// TwinCAT 3 PLC project Tc_SystemCx
// Title: Tc_SystemCx
// Company: NewEngineer
// Author: https://github.com/phucpha
// ProjectVersion: 0.0.0.1
// Description: This library expand of Tc2_systemCx
// ProgramVersion: 3.1.4024.0
// libraries:
//   Tc2_SystemCX, * (Beckhoff Automation GmbH)
//   Tc2_Utilities, * (Beckhoff Automation GmbH)
//   Tc3_Module, * (Beckhoff Automation GmbH)
// project tree:
//   / PlcTask.TcTTO
//   POUs/Cx70xx/ FB_Cx7_Read_EEPROM_CFIRM_KEY.TcPOU
//   Version/ Global_Version.TcGVL
// real-time tasks:
//   TASK PlcTask: cycle T#10ms, priority 20, ADS port 350

CONFIGURATION Tc_SystemCx
    RESOURCE PLC ON TwinCAT3
        TASK PlcTask(INTERVAL := T#10ms, PRIORITY := 20);
    END_RESOURCE
END_CONFIGURATION

// ---- Version/Global_Version.TcGVL
{attribute 'TcGenerated'}
{attribute 'no-analysis'}
{attribute 'linkalways'}
// This function has been automatically generated from the project information.
VAR_GLOBAL CONSTANT
	{attribute 'const_non_replaced'}
	stLibVersion_Tc_SystemCx : ST_LibVersion := (iMajor := 0, iMinor := 0, iBuild := 0, iRevision := 1, nFlags := 0, sVersion := '0.0.0.1');
END_VAR

// ---- POUs/Cx70xx/FB_Cx7_Read_EEPROM_CFIRM_KEY.TcPOU
{attribute 'hide_all_locals'}
FUNCTION_BLOCK FB_Cx7_Read_EEPROM_CFIRM_KEY
VAR_INPUT
	psKey: POINTER TO STRING(31);
END_VAR

VAR
	arrEEPRomRead : ARRAY [0..nSizeOfHASH_SHA512-1] OF BYTE;
	arrbHashGen : ARRAY [0..nSizeOfHASH_SHA512-1] OF BYTE;// Shouldn't edit it
// EEPROM
	bBusy            : BOOL;         // FB is working
    bEEpromError     : BOOL;         // FB has an Error
    nErrorID         : UDINT;        (* Error Code
    If nErrorID=DEVICE_INVALIDACCESS the EEPROM write cycles reached max. value. 
    If nErrorID=DEVICE_INVALIDPARM the given pointer parameter is invalid/null. 
    If nErrorID=DEVICE_INVALIDSIZE the given buffer size is too small or too big.
    If nErrorID=DEVICE_SRVNOTSUPP probably the image version need to be updated to support this feature. *)
    nDataSizeEEPROM  : UINT;         // current size of (read) EEPROM data in bytes (max.120 Bytes)
    nWritesCycles    : UINT;         // already performed EEPROM write cycles (maximum possible = 200)
	eRead 			 : UINT;
	fbRwEEPROM : FB_CX70xx_RW_EEPROM;
	bTmpCorrectKey : BOOL;
	idxLoop	: UINT;
END_VAR
VAR_OUTPUT
	bCorrectKey : BOOL;	
	bReadDone : BOOL;
END_VAR
VAR CONSTANT
	nSizeOfHASH_SHA512 : UINT := 64;// Shouldn't edit it
	nSizeOfKey : UINT := 32;// Shouldn't edit it
END_VAR

fbRwEEPROM(
		eMode          := E_CX70xx_EEPROM_Mode.ReadOnly,    // select RW mode
		pSrcBuf        := 0,        // pointer to WRITE EEPROM data buffer
		cbSrcBufSize   := 0,         // size of WRITE EEPROM data buffer (max.120 Bytes)
		pDstBuf        := ADR(arrEEPRomRead),        // pointer to READ EEPROM data buffer
		cbDstBufSize   := nSizeOfHASH_SHA512,         // max.size of READ EEPROM data buffer (max.120 Bytes)
		bBusy            => bBusy,         // FB is working
		bError           => bEEpromError,         // FB has an Error
		nErrorID         => nErrorID,        (* Error Code
		If nErrorID=DEVICE_INVALIDACCESS the EEPROM write cycles reached max. value. 
		If nErrorID=DEVICE_INVALIDPARM the given pointer parameter is invalid/null. 
		If nErrorID=DEVICE_INVALIDSIZE the given buffer size is too small or too big.
		If nErrorID=DEVICE_SRVNOTSUPP probably the image version need to be updated to support this feature. *)
		nDataSizeEEPROM  => nDataSizeEEPROM,        // current size of (read) EEPROM data in bytes (max.120 Bytes)
		nWritesCycles    => nWritesCycles         // already performed EEPROM write cycles (maximum possible = 200)
	);
CASE eRead OF
	0://Read
		fbRwEEPROM(bExecute := TRUE);
		IF NOT fbRwEEPROM.bBusy THEN
			eRead := 1;
		END_IF 
		bReadDone := FALSE;
	1:
		fbRwEEPROM(bExecute := FALSE);
		F_GenerateHashValue(
			hashMode := E_HashMode.HASH_SHA512,
			pData := psKey,
			nData := nSizeOfKey,
			pHash := ADR(arrbHashGen),
			nHash := nSizeOfHASH_SHA512
	); 
	bTmpCorrectKey := TRUE;
	FOR idxLoop := 0 TO nSizeOfHASH_SHA512-1 DO 
		IF arrbHashGen[idxLoop] <> arrEEPRomRead[idxLoop] THEN
			bTmpCorrectKey := FALSE;
		END_IF
	END_FOR
	bCorrectKey := bTmpCorrectKey;
	
END_CASE

END_FUNCTION_BLOCK
